// TIA Portal project "Conveyor Sorter" (V17)

(* hardware
DEVICE "S7-300/ET200M station_1"  S7-300 station
   slot 0: "Rail_0"  Rail  6ES7 390-1***0-0AA0
   slot 2: "PLC_1"  CPU 314C-2 PN/DP  6ES7 314-6EH04-0AB0  V3.3
      slot 2: "PROFINET interface_1"  PN-IO
         slot 1: "Port_1"  Port
         slot 2: "Port_2"  Port
      slot 5: "DI 24/DO 16_1"  DI24/DO16
      slot 6: "AI 5/AO 2_1"  AI5/AO2
      slot 7: "Count_1"  Counter
      slot 8: "Positioning_1"  Positioning
*)

// ===== PLC "PLC_1"  CPU 314C-2 PN/DP =====

VAR_GLOBAL   // PLC tag table "Default tag table"
   "FactoryIO_Running" AT %I0.0 : Bool;
   "Vision_Sensor1" AT %I0.1 : Bool;
   "Vision_Sensor2" AT %I0.2 : Bool;
   "Vision_Sensor3" AT %I0.3 : Bool;
   "PBL1" AT %I0.4 : Bool;
   "PFL1" AT %I0.5 : Bool;
   "PBL2" AT %I0.6 : Bool;
   "PFL2" AT %I0.7 : Bool;
   "PBL3" AT %I1.0 : Bool;
   "PFL3" AT %I1.1 : Bool;
   "START" AT %I1.2 : Bool;
   "STOP" AT %I1.3 : Bool;
   "RESET" AT %I1.4 : Bool;
   "Conveyor1" AT %Q0.0 : Bool;
   "Conveyor2" AT %Q0.1 : Bool;
   "Emitter" AT %Q0.2 : Bool;
   "Pusher1" AT %Q0.3 : Bool;
   "Pusher2" AT %Q0.4 : Bool;
   "Pusher3" AT %Q0.5 : Bool;
   "Green_Light" AT %Q0.6 : Bool;
   "Red_Light" AT %Q0.7 : Bool;
   "Yelloe_Light" AT %Q1.0 : Bool;
END_VAR

ORGANIZATION_BLOCK "OB1"   // OB1, LAD
{ S7_Optimized_Access := 'FALSE' }
VERSION : 0.1
   VAR_TEMP
      Temp_0 : Byte;
      Temp_1 : Byte;
      Temp_2 : Byte;
      Temp_3 : Byte;
      Temp_4 : Byte;
      Temp_5 : Byte;
      Temp_6 : Int;
      Temp_7 : Int;
      Temp_8 : Int;
      Temp_9 : Date_And_Time;
   END_VAR
BEGIN

REGION Network 1
   // Factory IO Main Switch
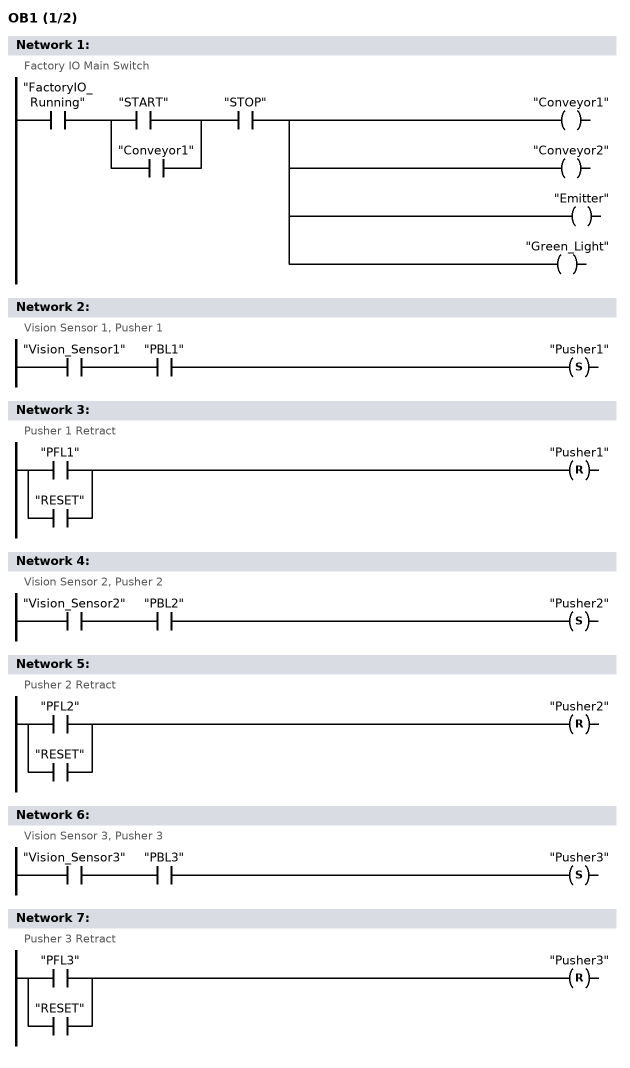
   RUNG wire#powerrail
      Contact( "FactoryIO_Running" )
      wire#w1
      Contact( "START" )
      wire#w2
      Contact( "STOP" )
      wire#w3
      Coil( "Conveyor1" )
   END_RUNG
   RUNG wire#w1
      Contact( "Conveyor1" )
   END_RUNG wire#w2
   RUNG wire#w3
      Coil( "Conveyor2" )
   END_RUNG
   RUNG wire#w3
      Coil( "Emitter" )
   END_RUNG
   RUNG wire#w3
      Coil( "Green_Light" )
   END_RUNG
   // the same network as SCL:
   "Conveyor1" := "FactoryIO_Running" AND ("START" OR "Conveyor1") AND "STOP";
   "Conveyor2" := "Conveyor1";
   "Emitter" := "Conveyor1";
   "Green_Light" := "Conveyor1";
END_REGION

REGION Network 2
   // Vision Sensor 1, Pusher 1
   RUNG wire#powerrail
      Contact( "Vision_Sensor1" )
      Contact( "PBL1" )
      S_Coil( "Pusher1" )
   END_RUNG
   // the same network as SCL:
   IF "Vision_Sensor1" AND "PBL1" THEN "Pusher1" := TRUE; END_IF;
END_REGION

REGION Network 3
   // Pusher 1 Retract
   RUNG wire#powerrail
      Contact( "PFL1" )
      wire#w1
      R_Coil( "Pusher1" )
   END_RUNG
   RUNG wire#powerrail
      Contact( "RESET" )
   END_RUNG wire#w1
   // the same network as SCL:
   IF "PFL1" OR "RESET" THEN "Pusher1" := FALSE; END_IF;
END_REGION

REGION Network 4
   // Vision Sensor 2, Pusher 2
   RUNG wire#powerrail
      Contact( "Vision_Sensor2" )
      Contact( "PBL2" )
      S_Coil( "Pusher2" )
   END_RUNG
   // the same network as SCL:
   IF "Vision_Sensor2" AND "PBL2" THEN "Pusher2" := TRUE; END_IF;
END_REGION

REGION Network 5
   // Pusher 2 Retract
   RUNG wire#powerrail
      Contact( "PFL2" )
      wire#w1
      R_Coil( "Pusher2" )
   END_RUNG
   RUNG wire#powerrail
      Contact( "RESET" )
   END_RUNG wire#w1
   // the same network as SCL:
   IF "PFL2" OR "RESET" THEN "Pusher2" := FALSE; END_IF;
END_REGION

REGION Network 6
   // Vision Sensor 3, Pusher 3
   RUNG wire#powerrail
      Contact( "Vision_Sensor3" )
      Contact( "PBL3" )
      S_Coil( "Pusher3" )
   END_RUNG
   // the same network as SCL:
   IF "Vision_Sensor3" AND "PBL3" THEN "Pusher3" := TRUE; END_IF;
END_REGION

REGION Network 7
   // Pusher 3 Retract
   RUNG wire#powerrail
      Contact( "PFL3" )
      wire#w1
      R_Coil( "Pusher3" )
   END_RUNG
   RUNG wire#powerrail
      Contact( "RESET" )
   END_RUNG wire#w1
   // the same network as SCL:
   IF "PFL3" OR "RESET" THEN "Pusher3" := FALSE; END_IF;
END_REGION

REGION Network 8
   // Stack light Red, when all conveyor are postive & Emitter Positive
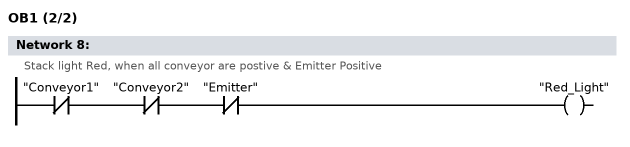
   RUNG wire#powerrail
      I_Contact( "Conveyor1" )
      I_Contact( "Conveyor2" )
      I_Contact( "Emitter" )
      Coil( "Red_Light" )
   END_RUNG
   // the same network as SCL:
   "Red_Light" := NOT "Conveyor1" AND NOT "Conveyor2" AND NOT "Emitter";
END_REGION
END_ORGANIZATION_BLOCK